TYPE CT_Track_BR_to_Tc_t :
STRUCT
    bStatus : BYTE;
    diError : DINT;
END_STRUCT
END_TYPE

(* stored: Version 1.1.0.1, ProductVersion 3.1.4024.6
   DUT CT_Track_BR_to_Tc_t: Id {d998620d-8bd2-44fc-8a31-d292ede48ec9} *)
